SUBAPPLICATION mapping_Softkeys_IX (* Mapping for all Softkey *)
  (* Standard: 61499-2 *)
  (* Version 1.0, 2023-01-29, Franz *)
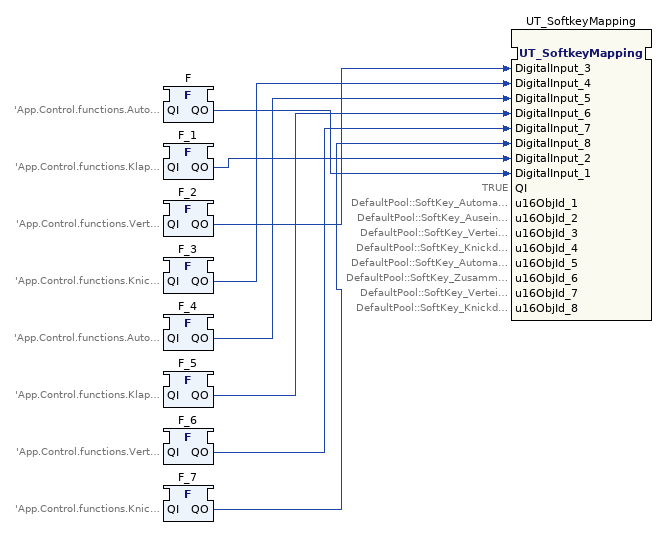
  FBS
    UT_SoftkeyMapping : UT_SoftkeyMapping(QI := TRUE, u16ObjId_1 := DefaultPool::SoftKey_Automatik_ein, u16ObjId_2 := DefaultPool::SoftKey_Auseinanderklappen, u16ObjId_3 := DefaultPool::SoftKey_Verteiler_senken, u16ObjId_4 := DefaultPool::SoftKey_Knickdeichsel_senken, u16ObjId_5 := DefaultPool::SoftKey_Automatik_aus, u16ObjId_6 := DefaultPool::SoftKey_Zusammenklappen, u16ObjId_7 := DefaultPool::SoftKey_Verteiler_heben, u16ObjId_8 := DefaultPool::SoftKey_Knickdeichsel_heben);
  END_FBS
  SUBAPPS
    F : F(QI := 'App.Control.functions.Automatik.ein.SoftKey');
    F_1 : F(QI := 'App.Control.functions.Klappen.SoftKey_heben.IX');
    F_2 : F(QI := 'App.Control.functions.Verteiler.SoftKey_senken.IX');
    F_3 : F(QI := 'App.Control.functions.Knickdeichsel.SoftKey_senken.IX');
    F_4 : F(QI := 'App.Control.functions.Automatik.aus.SoftKey');
    F_5 : F(QI := 'App.Control.functions.Klappen.SoftKey_senken.IX');
    F_6 : F(QI := 'App.Control.functions.Verteiler.SoftKey_heben.IX');
    F_7 : F(QI := 'App.Control.functions.Knickdeichsel.SoftKey_heben.IX');
  END_SUBAPPS
  DATA_CONNECTIONS
    F_2.QO TO UT_SoftkeyMapping.DigitalInput_3;
    F_3.QO TO UT_SoftkeyMapping.DigitalInput_4;
    F_4.QO TO UT_SoftkeyMapping.DigitalInput_5;
    F_5.QO TO UT_SoftkeyMapping.DigitalInput_6;
    F_6.QO TO UT_SoftkeyMapping.DigitalInput_7;
    F_7.QO TO UT_SoftkeyMapping.DigitalInput_8;
    F_1.QO TO UT_SoftkeyMapping.DigitalInput_2;
    F.QO TO UT_SoftkeyMapping.DigitalInput_1;
  END_CONNECTIONS
END_SUBAPPLICATION
